(* PLC project test_slave, lolitech beremiz 1 *)
(* stored: creationDateTime 2008-06-24 18:44:00, modificationDateTime 2008-06-27 15:41:26, language en-US *)

PROGRAM test_main
  VAR
    PLC_OUT AT %QW0.0.3.8193.0 : INT;
    PLC_IN AT %IW0.0.3.8192.0 : INT;
  END_VAR

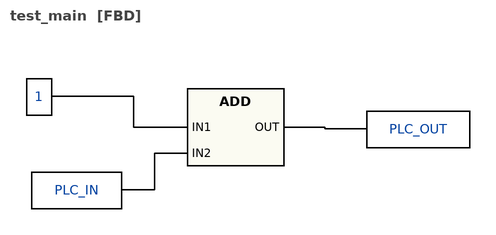
(* FBD diagram, written out as Structured Text *)
PLC_OUT := 1 + PLC_IN;
END_PROGRAM

CONFIGURATION conf
  RESOURCE res ON PLC
    TASK tache(INTERVAL := 00:00:00.050000, PRIORITY := 0);
    PROGRAM toto WITH tache : test_main;
  END_RESOURCE
END_CONFIGURATION
